ABB RobotStudio station: OefenTCP.rsstnx

Station OefenTCP (saved by RobotStudio 23.3.10550.0)
Controller IRB120_3_58
  mechanical unit ROB_1: IRB120_3_58__01, 6 joints, base frame (0, 0, 0) mm
Layout (positions relative to the parent item):
  - tSpintec [mechanism] at (364.35, 0, 594) mm, rotated rx 180 ry 60 rz 180 deg
      TCP tSpintec at (31.79, 0, 229.64) mm, rotated rx 0 ry 38 rz 0 deg
      links: SpintecTool
  - IRB120_3_58__01 [mechanism, from %ABB.RobotStudio.Models.IRB120%\IRB120_3_58_G_01.rslib] at (0, 0, 0) mm; joint values [0, 0, 0, 0, 0.5236, 0] (rad or m)
  - Frame_4 [frame] at (31.79, 0, 229.64) mm, rotated rx 0 ry 38 rz 0 deg
Attachment: tSpintec is attached to IRB120_3_58__01 / Link6
Targets, tools, work objects and paths stored in the station, written as RAPID:
! task T_ROB1
MODULE CalibData
  PERS tooldata tSpintec:=[TRUE,[[31.793,0,229.639],[0.945518576,0,0.325568154,0]],[1,[-73.579,279.02,0],[1,0,0,0],0,0,0]];
ENDMODULE

